FUNCTION TryConvert_TIME_TO_TIME : BOOL
VAR_INPUT
	in : TIME;
	out : REFERENCE TO TIME;
END_VAR

out := in;
TryConvert_TIME_TO_TIME := TRUE;

END_FUNCTION

(* stored: Version 1.1.0.1, ProductVersion 3.1.4024.12
   POU TryConvert_TIME_TO_TIME: Id {2e45ff33-a23b-4124-995d-7d5d63c69e24}, SpecialFunc None *)
